PROGRAM MAIN
VAR
    a
END_VAR

END_PROGRAM

(* stored: Version 1.1.0.1, ProductVersion 3.1.4024.3
   POU MAIN: Id {54cec01d-530e-47bf-9e74-86ce6ef45a25}, SpecialFunc None *)
